(* CoDeSys 2.3 export: SINUSFUNCTION.EXP *)

(* POU SinusFunction, ST *)
FUNCTION SinusFunction : REAL
VAR_INPUT
	t	:	REAL;		(*Input Time*)
END_VAR
VAR
	w	:	REAL := 1; 	(*Frequency*)
	A	:	REAL := 1;	(*Amplitude*)
	offs:	REAL := 0;	(*Offset*)
END_VAR
(*Generate Sine-Wave*)
SinusFunction := A*SIN(w*t) + offs;
END_FUNCTION
